// TwinCAT 3 PLC project Main
// ProgramVersion: 3.1.4024.0
// libraries:
//   Tc2_Standard, * (Beckhoff Automation GmbH)
//   Tc2_System, * (Beckhoff Automation GmbH)
//   Tc3_Module, * (Beckhoff Automation GmbH)
//   TcUnit,1.2.0.0,www.tcunit.org
// project tree:
//   GVLs/ GVL_IO.TcGVL
//   / PlcTask.TcTTO, Task_Test.TcTTO
//   POUs/ FB_MotorControl.TcPOU, MAIN.TcPOU
//   UnitTest/ FB_MotorControl_Test.TcPOU, UnitTestProgram.TcPOU
// real-time tasks:
//   TASK PlcTask: cycle T#10ms, priority 20, ADS port 350
//   TASK Task_Test: cycle T#10ms, priority 1, ADS port 351

CONFIGURATION Main
    RESOURCE PLC ON TwinCAT3
        TASK PlcTask(INTERVAL := T#10ms, PRIORITY := 20);
        TASK Task_Test(INTERVAL := T#10ms, PRIORITY := 1);
        PROGRAM MAIN WITH PlcTask : MAIN;
        PROGRAM UnitTestProgram WITH Task_Test : UnitTestProgram;
    END_RESOURCE
END_CONFIGURATION

// ---- GVLs/GVL_IO.TcGVL
{attribute 'qualified_only'}
VAR_GLOBAL
	Button1 AT %I* : BOOL;
	Button2 AT %I* : BOOL;
	Sensor AT %I* : BOOL;
	Motor AT %Q* : BOOL;	
END_VAR

// ---- POUs/MAIN.TcPOU
PROGRAM MAIN
VAR
	MotorControl : FB_MotorControl;
END_VAR

MotorControl( button1 := GVL_IO.Button1,
	          button2 := GVL_IO.Button2,
	          sensor := GVL_IO.Sensor,
			  Motor => GVL_IO.Motor);

END_PROGRAM

// ---- POUs/FB_MotorControl.TcPOU
FUNCTION_BLOCK FB_MotorControl
VAR_INPUT
	Button1 : BOOL;
	Button2 : BOOL;
	Sensor : BOOL;
END_VAR
VAR_OUTPUT
	Motor : BOOL;
END_VAR
VAR
END_VAR

Motor := IsMotorTurnedOn(Button1, Button2, Sensor);

METHOD IsMotorTurnedOn : BOOL
VAR_INPUT
	button1 : BOOL;
	button2 : BOOL;
	sensor : bool;
END_VAR
IsMotorTurnedOn := button1 AND button2 AND NOT sensor;
END_METHOD

END_FUNCTION_BLOCK

// ---- UnitTest/UnitTestProgram.TcPOU
PROGRAM UnitTestProgram
VAR
	MotorControl_Test : FB_MotorControl_Test;
END_VAR

TcUnit.RUN();

END_PROGRAM

// ---- UnitTest/FB_MotorControl_Test.TcPOU
FUNCTION_BLOCK FB_MotorControl_Test EXTENDS FB_TestSuite
VAR_INPUT
END_VAR
VAR_OUTPUT
END_VAR
VAR
END_VAR

TestWhenSensorIsOff();
TestWhenButton1Off();

METHOD TestWhenButton1Off
VAR_INPUT
END_VAR
VAR
	motorControl : FB_MotorControl;
	result : BOOL;
	expected_result : BOOL := TRUE;
	
END_VAR
TEST('TestWhenButton1Off');

motorControl( Button1 := FALSE, Button2 := TRUE, Sensor := FALSE, Motor => result);


AssertEquals(Expected := expected_result,
             Actual := result,
             Message := 'The output is not correct' );

TEST_FINISHED();
END_METHOD

METHOD TestWhenSensorIsOff
VAR_INPUT
END_VAR
VAR
	motorControl : FB_MotorControl;
	result : BOOL;
	expected_result : BOOL := TRUE;
END_VAR
TEST('TestWhenSensorIsOff');

motorControl( Button1 := TRUE, Button2 := TRUE, Sensor := FALSE, Motor => result);
 
AssertEquals(Expected := expected_result,
             Actual := result,
             Message := 'The output is not correct' );
TEST_FINISHED();
END_METHOD

END_FUNCTION_BLOCK
